// Returns information about the variable as ST_VarInfo.
FUNCTION F_GetVarInfo : ST_VarInfo
VAR_INPUT
	variable	: ANY;	// Variable to get the inforation from
END_VAR
VAR
END_VAR

F_GetVarInfo.Address := variable.pValue;
F_GetVarInfo.DataType := variable.TypeClass;
F_GetVarInfo.Size := DINT_TO_UDINT(variable.diSize);

END_FUNCTION

(* stored: Version 1.1.0.1, ProductVersion 3.1.4024.14
   POU F_GetVarInfo: Id {428533f5-71b2-08f8-0455-adf25c0fe5b3}, SpecialFunc None *)
